{attribute addProperty BoxType "EL3102-0000-0016"}
{attribute addProperty Id "StatusAT %I*Status_F9B4A013587.251ValueAT %I*INT16217"}
{attribute addProperty CRC "2269758005"}
{attribute addProperty SizeInBites "74"}
{attribute addProperty SizeInBytes "9.25"}
TYPE AI_Standard_Channel_8749C235 :
STRUCT
	{attribute addProperty Name "Status"}
	Status AT %I* : Status_F9B4A013;
	{attribute addProperty Name "Value"}
	Value AT %I* : INT;
END_STRUCT
END_TYPE

(* stored: Version 1.2.0.0, ProductVersion 3.1.4024.9
   DUT AI_Standard_Channel_8749C235: Id {9e66ffe4-8fb3-40c6-acb7-12ef67e637a7} *)
